PROGRAM Axis05_Interlock
VAR
//System_Bit
	Always_ON	:	BOOL	:=TRUE	;//상시 ON 
	Always_OFF	:	BOOL	:=FALSE	;//상시 OFF
END_VAR
VAR // added by the converter: edge detectors and wires of the graphical bodies
    _w1, _w2 : BOOL;
END_VAR

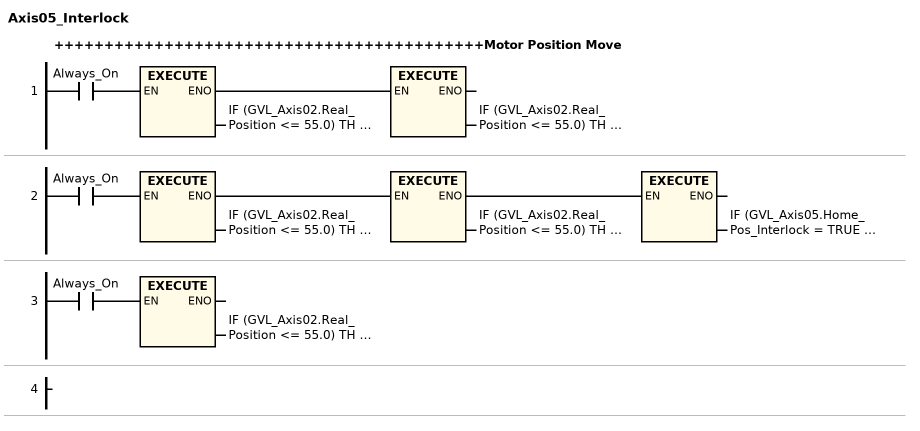
// NETWORK 1: +++++++++++++++++++++++++++++++++++++++++++Motor Position Move
_w1 := Always_On;
IF _w1 THEN
    IF (GVL_Axis02.Real_Position <= 55.0) THEN
        GVL_Axis05.Home_Pos_Interlock := TRUE;
    ELSE
        IF (GVL_Axis05.Home_Position_Data >= -10) AND 
           (GVL_Axis05.Home_Position_Data <= 10) THEN
            GVL_Axis05.Home_Pos_Interlock := TRUE;
        ELSE 
           GVL_Axis05.Home_Pos_Interlock := FALSE;
        END_IF;
    END_IF;
END_IF
IF _w1 THEN
    IF (GVL_Axis02.Real_Position <= 55.0) THEN
        GVL_Axis05.Wait_Pos_Interlock := TRUE;
    ELSE
        IF (GVL_Axis05.Wait_Position_Data >= -10) AND 
           (GVL_Axis05.Wait_Position_Data <= 10) THEN
            GVL_Axis05.Wait_Pos_Interlock := TRUE;
        ELSE 
           GVL_Axis05.Wait_Pos_Interlock := FALSE;
        END_IF;
    END_IF;
END_IF

// NETWORK 2
_w2 := Always_On;
IF _w2 THEN
    IF (GVL_Axis02.Real_Position <= 55.0) THEN
        GVL_Axis05.Target_Pos_Interlock := TRUE;
    ELSE
        IF (GVL_Axis05.Target_Position_Data >= -10) AND 
           (GVL_Axis05.Target_Position_Data <= 10) THEN
            GVL_Axis05.Target_Pos_Interlock := TRUE;
        ELSE 
           GVL_Axis05.Target_Pos_Interlock := FALSE;
        END_IF;
    END_IF;
END_IF
IF _w2 THEN
    IF (GVL_Axis02.Real_Position <= 55.0) THEN
        GVL_Axis05.Work_End_Pos_Interlock := TRUE;
    ELSE
        IF (GVL_Axis05.Work_End_Position_Data >= -10) AND 
           (GVL_Axis05.Work_End_Position_Data <= 10) THEN
            GVL_Axis05.Work_End_Pos_Interlock := TRUE;
        ELSE 
           GVL_Axis05.Work_End_Pos_Interlock := FALSE;
        END_IF;
    END_IF;
END_IF
IF _w2 THEN
    IF (GVL_Axis05.Home_Pos_Interlock = TRUE) AND (GVL_Axis05.Wait_Pos_Interlock = TRUE) AND (GVL_Axis05.Target_Pos_Interlock = TRUE) AND (GVL_Axis05.Work_End_POs_Interlock = TRUE) THEN
    	GVL_Axis05.Interlock := TRUE;
    	ELSE
    	GVL_Axis05.Interlock := FALSE;	
    
    END_IF
END_IF

// NETWORK 3
IF Always_On THEN
    IF (GVL_Axis02.Real_Position <= 55.0) THEN
        GVL_Axis05.Home_ORG_Interlock := TRUE;
    ELSE
           GVL_Axis05.Home_ORG_Interlock := FALSE;
    END_IF;
END_IF

// NETWORK 4

END_PROGRAM

(* stored: Version 1.1.0.1, ProductVersion 3.1.4024.15
   POU Axis05_Interlock: Id {baa90fa8-6f44-44e8-8b25-6afdea8e539e}, SpecialFunc None *)
